// TIA Portal V20 export
TYPE "LER_typeCommonDataStackMotion"
// stored: Access Published
   STRUCT
      MotionToPLC : "LER_typeMotionToPLC";
   END_STRUCT;
END_TYPE
